// TIA Portal project "FactoryIO_Template_S7-1500_V15_V16_V17" (V17)

(* hardware
DEVICE "S71500/ET200MP-Station_1"  S7-1500 station
   slot 0: "Profilschiene_0"  6ES7 590-1***0-0AA0
   slot 1: "PLC_1"  CPU 1511-1 PN  6ES7 511-1AK00-0AB0  V1.8
   slot 2: "DI 16x24VDC BA_1"  DI 16x24VDC BA  6ES7 521-1BH10-0AA0  V1.0
   slot 3: "DQ 32x24VDC/0.5A BA_1"  DQ 32x24VDC/0.5A BA  6ES7 522-1BL10-0AA0  V1.1
*)

// ===== PLC "PLC_1"  CPU 1511-1 PN =====

VAR_GLOBAL   // PLC tag table "Standard-Variablentabelle"
   "Tag_1" AT %E0.0 : Bool;
   "Tag_3" AT %E0.1 : Bool;
   "ALWAYS_FALSE" AT %M100.1 : Bool;
END_VAR

VAR_GLOBAL   // PLC tag table "R00_S01_DI"
   "PALLET_AT_ENTRY" AT %I10.0 : Bool;
   "PALLET_AT_EXIT" AT %I10.1 : Bool;
   "PALLET_LOADED" AT %I10.2 : Bool;
   "BOX_AT_ENTRY" AT %I10.3 : Bool;
   "PUSHER_LIMIT" AT %I10.4 : Bool;
   "PLATE_LIMIT" AT %I10.5 : Bool;
   "CLAMPED" AT %I10.6 : Bool;
   "ELEVATOR_MOVING" AT %I10.7 : Bool;
   "START" AT %I11.0 : Bool;
   "RESET" AT %I11.1 : Bool;
   "STOP" AT %I11.2 : Bool;
   "EMERGENCY_STOP" AT %I11.3 : Bool;
   "AUTO" AT %I11.4 : Bool;
   "FACTORY_IO_RUNING" AT %I11.5 : Bool;
END_VAR

VAR_GLOBAL   // PLC tag table "R00_S02_D0"
   "PALLET_FEEDER" AT %A0.0 : Bool;
   "LOAD_PALLET" AT %Q0.1 : Bool;
   "EXIT_CONVEYOR" AT %Q0.2 : Bool;
   "MOVE_TO_LIMIT" AT %Q0.3 : Bool;
   "ELEVATOR_UP" AT %Q0.4 : Bool;
   "ELEVATOR_DOWN" AT %Q0.5 : Bool;
   "BOX_FEEDER" AT %Q0.6 : Bool;
   "TURN" AT %Q0.7 : Bool;
   "PUSH" AT %Q1.0 : Bool;
   "LOAD_BELT" AT %Q1.1 : Bool;
   "CLAMP" AT %Q1.2 : Bool;
   "OPEN_PLATE" AT %Q1.3 : Bool;
   "WARNING_LIGHT" AT %Q1.4 : Bool;
   "START_LIGHT" AT %Q1.5 : Bool;
   "RESET_LIGHT" AT %Q1.6 : Bool;
   "STOP_LIGHT" AT %Q1.7 : Bool;
END_VAR

DATA_BLOCK "CONTADOR_CAJAS"   // DB2
{ S7_Optimized_Access := 'TRUE' }
VERSION : 0.1
   VAR
      RESET_CONTADOR_CAJAS_EN_FILA : Bool;
      FILA_COMPLETA : Bool;
      P_FILA_COMPLETA : Bool;
      RESET_NUM_FILAS : Bool;
      NIVEL_COMPLETO : Bool;
      P_NIVEL_COMPLETO : Bool;
      CANTIDAD_MAXIMA_NIVELES : Int := 4;
      RESET_NUM_NIVELES : Bool;
      CANTIDAD_MAXIMA_CAJAS_POR_FILA : Int := 3;
      CANTIDAD_MAXIMA_FILAS_POR_NIVEL : Int;
   END_VAR
BEGIN
END_DATA_BLOCK

DATA_BLOCK "PALETIZADORA_AUTOMATICO_DB"   // DB5
{ S7_Optimized_Access := 'TRUE' }
VERSION : 0.1
// stored: InstanceOfName PALETIZADORA_AUTOMATICO
"PALETIZADORA_AUTOMATICO"
BEGIN
END_DATA_BLOCK

// folder: System blocks/Program resources

DATA_BLOCK "CONTADOR_CAJAS_EN_FILA"   // DB1
{ S7_Optimized_Access := 'TRUE' }
AUTHOR : Simatic
FAMILY : IEC
NAME : CNTR
VERSION : 1.0
// stored: InstanceOfName IEC_COUNTER
"IEC_COUNTER"
BEGIN
END_DATA_BLOCK

DATA_BLOCK "CONTADOR_FILAS"   // DB3
{ S7_Optimized_Access := 'TRUE' }
AUTHOR : Simatic
FAMILY : IEC
NAME : CNTR
VERSION : 1.0
// stored: InstanceOfName IEC_COUNTER
"IEC_COUNTER"
BEGIN
END_DATA_BLOCK

DATA_BLOCK "CONTADOR_NIVELES"   // DB4
{ S7_Optimized_Access := 'TRUE' }
AUTHOR : Simatic
FAMILY : IEC
NAME : CNTR
VERSION : 1.0
// stored: InstanceOfName IEC_COUNTER
"IEC_COUNTER"
BEGIN
END_DATA_BLOCK

// folder: (top level)

FUNCTION_BLOCK "PALETIZADORA_AUTOMATICO"   // FB1, GRAPH_PLUS
{ S7_Optimized_Access := 'TRUE' }
VERSION : 0.1
   VAR_INPUT
      OFF_SQ : Bool := false;   // Turn sequence off
      INIT_SQ : Bool := false;   // Set sequence to initial state
      ACK_EF : Bool := false;   // Acknowledge all errors and faults
      S_PREV : Bool := false;   // Output previous step in parameter S_NO
      S_NEXT : Bool := false;   // Indicate next step in parameter S_NO
      SW_AUTO : Bool := false;   // Automatic mode
      SW_TAP : Bool := false;   // Semiautomatic/switch with transition
      SW_TOP : Bool := false;   // Semiautomatic/ignore transition
      SW_MAN : Bool := false;   // Manual mode
      S_SEL : Int := 0;   // Select step to be output to S_NO
      S_ON : Bool := false;   // Activate step indicated in S_NO
      S_OFF : Bool := false;   // Deactivate step indicated S_NO
      T_PUSH : Bool := false;   // Enable transition to switch in semi automatic mode
   END_VAR
   VAR_OUTPUT
      S_NO : Int := 0;   // Step number
      S_MORE : Bool := false;   // More steps are available and can be shown in S_NO
      S_ACTIVE : Bool := false;   // Step indicated in S_NO is active
      ERR_FLT : Bool := false;   // Interlock or supervision group error
      AUTO_ON : Bool := false;   // Automatic mode is active
      TAP_ON : Bool := false;   // Semiautomatic mode/step with transition enabled
      TOP_ON : Bool := false;   // Semiautomatic mode/ignore transition enabled
      MAN_ON : Bool := false;   // Manual mode is active
   END_VAR
   VAR
      HMI_INFO : Array[0..8] of UInt;
      IF_PAR : G7_IfParPlus_V2;
      RT_DATA : G7_RTDataPlus_V2;   // Internal data area
      Trans1 : G7_TransitionPlus_V2;   // Transition structure
      Trans2 : G7_TransitionPlus_V2;   // Transition structure
      Trans3 : G7_TransitionPlus_V2;   // Transition structure
      Trans4 : G7_TransitionPlus_V2;   // Transition structure
      Trans5 : G7_TransitionPlus_V2;   // Transition structure
      Trans6 : G7_TransitionPlus_V2;   // Transition structure
      Trans7 : G7_TransitionPlus_V2;   // Transition structure
      Trans8 : G7_TransitionPlus_V2;   // Transition structure
      Trans9 : G7_TransitionPlus_V2;   // Transition structure
      Trans10 : G7_TransitionPlus_V2;   // Transition structure
      Trans11 : G7_TransitionPlus_V2;   // Transition structure
      Trans12 : G7_TransitionPlus_V2;   // Transition structure
      Trans14 : G7_TransitionPlus_V2;   // Transition structure
      Trans13 : G7_TransitionPlus_V2;   // Transition structure
      Trans15 : G7_TransitionPlus_V2;   // Transition structure
      Trans16 : G7_TransitionPlus_V2;   // Transition structure
      Trans17 : G7_TransitionPlus_V2;   // Transition structure
      Trans18 : G7_TransitionPlus_V2;   // Transition structure
      Trans19 : G7_TransitionPlus_V2;   // Transition structure
      Trans20 : G7_TransitionPlus_V2;   // Transition structure
      START : G7_StepPlus_V2;   // Step structure
      LOAD_PALLET : G7_StepPlus_V2;   // Step structure
      STOP_PALLET : G7_StepPlus_V2;   // Step structure
      EL_UP_TO_TOP : G7_StepPlus_V2;   // Step structure
      BOX_FEEDER : G7_StepPlus_V2;   // Step structure
      WAIT_1 : G7_StepPlus_V2;   // Step structure
      PUSH_N_PART : G7_StepPlus_V2;   // Step structure
      INTER : G7_StepPlus_V2;   // Step structure
      N_FILAS_IMPAR : G7_StepPlus_V2;   // Step structure
      CLAMP : G7_StepPlus_V2;   // Step structure
      TURN_ON : G7_StepPlus_V2;   // Step structure
      TURN_OFF : G7_StepPlus_V2;   // Step structure
      OPENPLATE : G7_StepPlus_V2;   // Step structure
      ELEVATOR_DOWN : G7_StepPlus_V2;   // Step structure
      ELEVATOR_DOWN_TO_BOTTON : G7_StepPlus_V2;   // Step structure
      EXIT_CONVEYOR : G7_StepPlus_V2;   // Step structure
      SINI : Array[0..1] of USInt;
      LSTT : Array[0..19] of USInt;
      ATAJ : Array[0..19] of USInt;
      ATAB : Array[0..19] of USInt;
      PSTT : Array[0..19] of USInt;
      NSTT : Array[0..19] of USInt;
      ASSJ : Array[0..15] of USInt;
      ASSB : Array[0..15] of USInt;
      PTTS : Array[0..15] of USInt;
      NTTS : Array[0..15] of USInt;
      SW_SQTS : Array[0..15] of USInt;
      SWITCH : Array[0..6] of USInt;
      TVX : Array[0..9] of USInt;
      TTX : Array[0..9] of USInt;
      TSX : Array[0..1] of USInt;
      S00X : Array[0..1] of USInt;
      SOFFX : Array[0..1] of USInt;
      SONX : Array[0..1] of USInt;
      SAX : Array[0..1] of USInt;
      SERRX : Array[0..16] of USInt;
      SMX : Array[0..16] of USInt;
      S0X : Array[0..16] of USInt;
      S1X : Array[0..16] of USInt;
      IL_ALARM_INST : Program_Alarm;
      SUP_ALARM_INST : Program_Alarm;
      STEP_TIME_ALARM_INST : Program_Alarm;
      IEC_TIMER_INST : IEC_TIMER;
      TRANSACTION_FLAG : Bool := false;
   END_VAR
   // SINI[0] := 2;
   // LSTT[0] := 255;
   // LSTT[1] := 255;
   // LSTT[2] := 255;
   // LSTT[3] := 255;
   // LSTT[4] := 255;
   // LSTT[5] := 255;
   // LSTT[6] := 255;
   // LSTT[8] := 255;
   // LSTT[9] := 4;
   // LSTT[10] := 255;
   // LSTT[11] := 255;
   // LSTT[12] := 255;
   // LSTT[13] := 255;
   // LSTT[14] := 255;
   // LSTT[15] := 255;
   // LSTT[16] := 4;
   // LSTT[17] := 255;
   // LSTT[18] := 255;
   // ATAJ[1] := 1;
   // ATAJ[2] := 2;
   // ATAJ[3] := 3;
   // ATAJ[4] := 4;
   // ATAJ[5] := 5;
   // ATAJ[6] := 6;
   // ATAJ[7] := 7;
   // ATAJ[8] := 8;
   // ATAJ[9] := 9;
   // ATAJ[10] := 10;
   // ATAJ[11] := 11;
   // ATAJ[12] := 12;
   // ATAJ[13] := 14;
   // ATAJ[14] := 13;
   // ATAJ[15] := 15;
   // ATAJ[16] := 16;
   // ATAJ[17] := 17;
   // ATAJ[18] := 18;
   // ATAJ[19] := 19;
   // ATAB[1] := 1;
   // ATAB[2] := 2;
   // ATAB[3] := 3;
   // ATAB[4] := 4;
   // ATAB[5] := 5;
   // ATAB[6] := 6;
   // ATAB[7] := 8;
   // ATAB[8] := 7;
   // ATAB[9] := 10;
   // ATAB[10] := 9;
   // ATAB[11] := 12;
   // ATAB[12] := 11;
   // ATAB[13] := 13;
   // ATAB[14] := 14;
   // ATAB[15] := 15;
   // ATAB[16] := 17;
   // ATAB[17] := 16;
   // ATAB[18] := 18;
   // ATAB[19] := 19;
   // PSTT[1] := 1;
   // PSTT[2] := 2;
   // PSTT[3] := 3;
   // PSTT[4] := 4;
   // PSTT[5] := 5;
   // PSTT[6] := 6;
   // PSTT[7] := 7;
   // PSTT[8] := 7;
   // PSTT[9] := 8;
   // PSTT[10] := 8;
   // PSTT[11] := 9;
   // PSTT[12] := 9;
   // PSTT[13] := 10;
   // PSTT[14] := 11;
   // PSTT[15] := 12;
   // PSTT[16] := 13;
   // PSTT[17] := 13;
   // PSTT[18] := 14;
   // PSTT[19] := 15;
   // NSTT[0] := 1;
   // NSTT[1] := 2;
   // NSTT[2] := 3;
   // NSTT[3] := 4;
   // NSTT[4] := 5;
   // NSTT[5] := 6;
   // NSTT[6] := 7;
   // NSTT[8] := 8;
   // NSTT[9] := 4;
   // NSTT[10] := 9;
   // NSTT[11] := 10;
   // NSTT[12] := 11;
   // NSTT[13] := 12;
   // NSTT[14] := 12;
   // NSTT[15] := 13;
   // NSTT[16] := 4;
   // NSTT[17] := 14;
   // NSTT[18] := 15;
   // ASSJ[1] := 1;
   // ASSJ[2] := 2;
   // ASSJ[3] := 3;
   // ASSJ[4] := 4;
   // ASSJ[5] := 5;
   // ASSJ[6] := 6;
   // ASSJ[7] := 7;
   // ASSJ[8] := 8;
   // ASSJ[9] := 9;
   // ASSJ[10] := 10;
   // ASSJ[11] := 11;
   // ASSJ[12] := 12;
   // ASSJ[13] := 13;
   // ASSJ[14] := 14;
   // ASSJ[15] := 15;
   // ASSB[1] := 1;
   // ASSB[2] := 2;
   // ASSB[3] := 3;
   // ASSB[4] := 4;
   // ASSB[5] := 5;
   // ASSB[6] := 6;
   // ASSB[7] := 7;
   // ASSB[8] := 8;
   // ASSB[9] := 9;
   // ASSB[10] := 10;
   // ASSB[11] := 11;
   // ASSB[12] := 12;
   // ASSB[13] := 13;
   // ASSB[14] := 14;
   // ASSB[15] := 15;
   // PTTS[0] := 255;
   // PTTS[2] := 1;
   // PTTS[3] := 2;
   // PTTS[4] := 3;
   // PTTS[5] := 4;
   // PTTS[6] := 5;
   // PTTS[7] := 6;
   // PTTS[8] := 8;
   // PTTS[9] := 10;
   // PTTS[10] := 11;
   // PTTS[11] := 12;
   // PTTS[12] := 13;
   // PTTS[13] := 15;
   // PTTS[14] := 17;
   // PTTS[15] := 18;
   // NTTS[1] := 1;
   // NTTS[2] := 2;
   // NTTS[3] := 3;
   // NTTS[4] := 4;
   // NTTS[5] := 5;
   // NTTS[6] := 6;
   // NTTS[7] := 7;
   // NTTS[8] := 9;
   // NTTS[9] := 11;
   // NTTS[10] := 13;
   // NTTS[11] := 14;
   // NTTS[12] := 15;
   // NTTS[13] := 16;
   // NTTS[14] := 18;
   // NTTS[15] := 19;
   // SW_SQTS[8] := 1;
   // SW_SQTS[9] := 2;
   // SW_SQTS[10] := 3;
   // SW_SQTS[11] := 4;
   // SW_SQTS[12] := 5;
   // SW_SQTS[13] := 5;
   // SW_SQTS[14] := 6;
   // SW_SQTS[15] := 6;
   // TVX[0] := 16#1;
   // TTX[0] := 16#1;
   // TSX[0] := 16#1;
   // S00X[0] := 16#1;
   // SOFFX[0] := 16#1;
   // SONX[0] := 16#1;
   // SAX[0] := 16#1;
   // SERRX[0] := 16#1;
   // SMX[0] := 16#1;
   // S0X[0] := 16#1;
   // S1X[0] := 16#1;
BEGIN
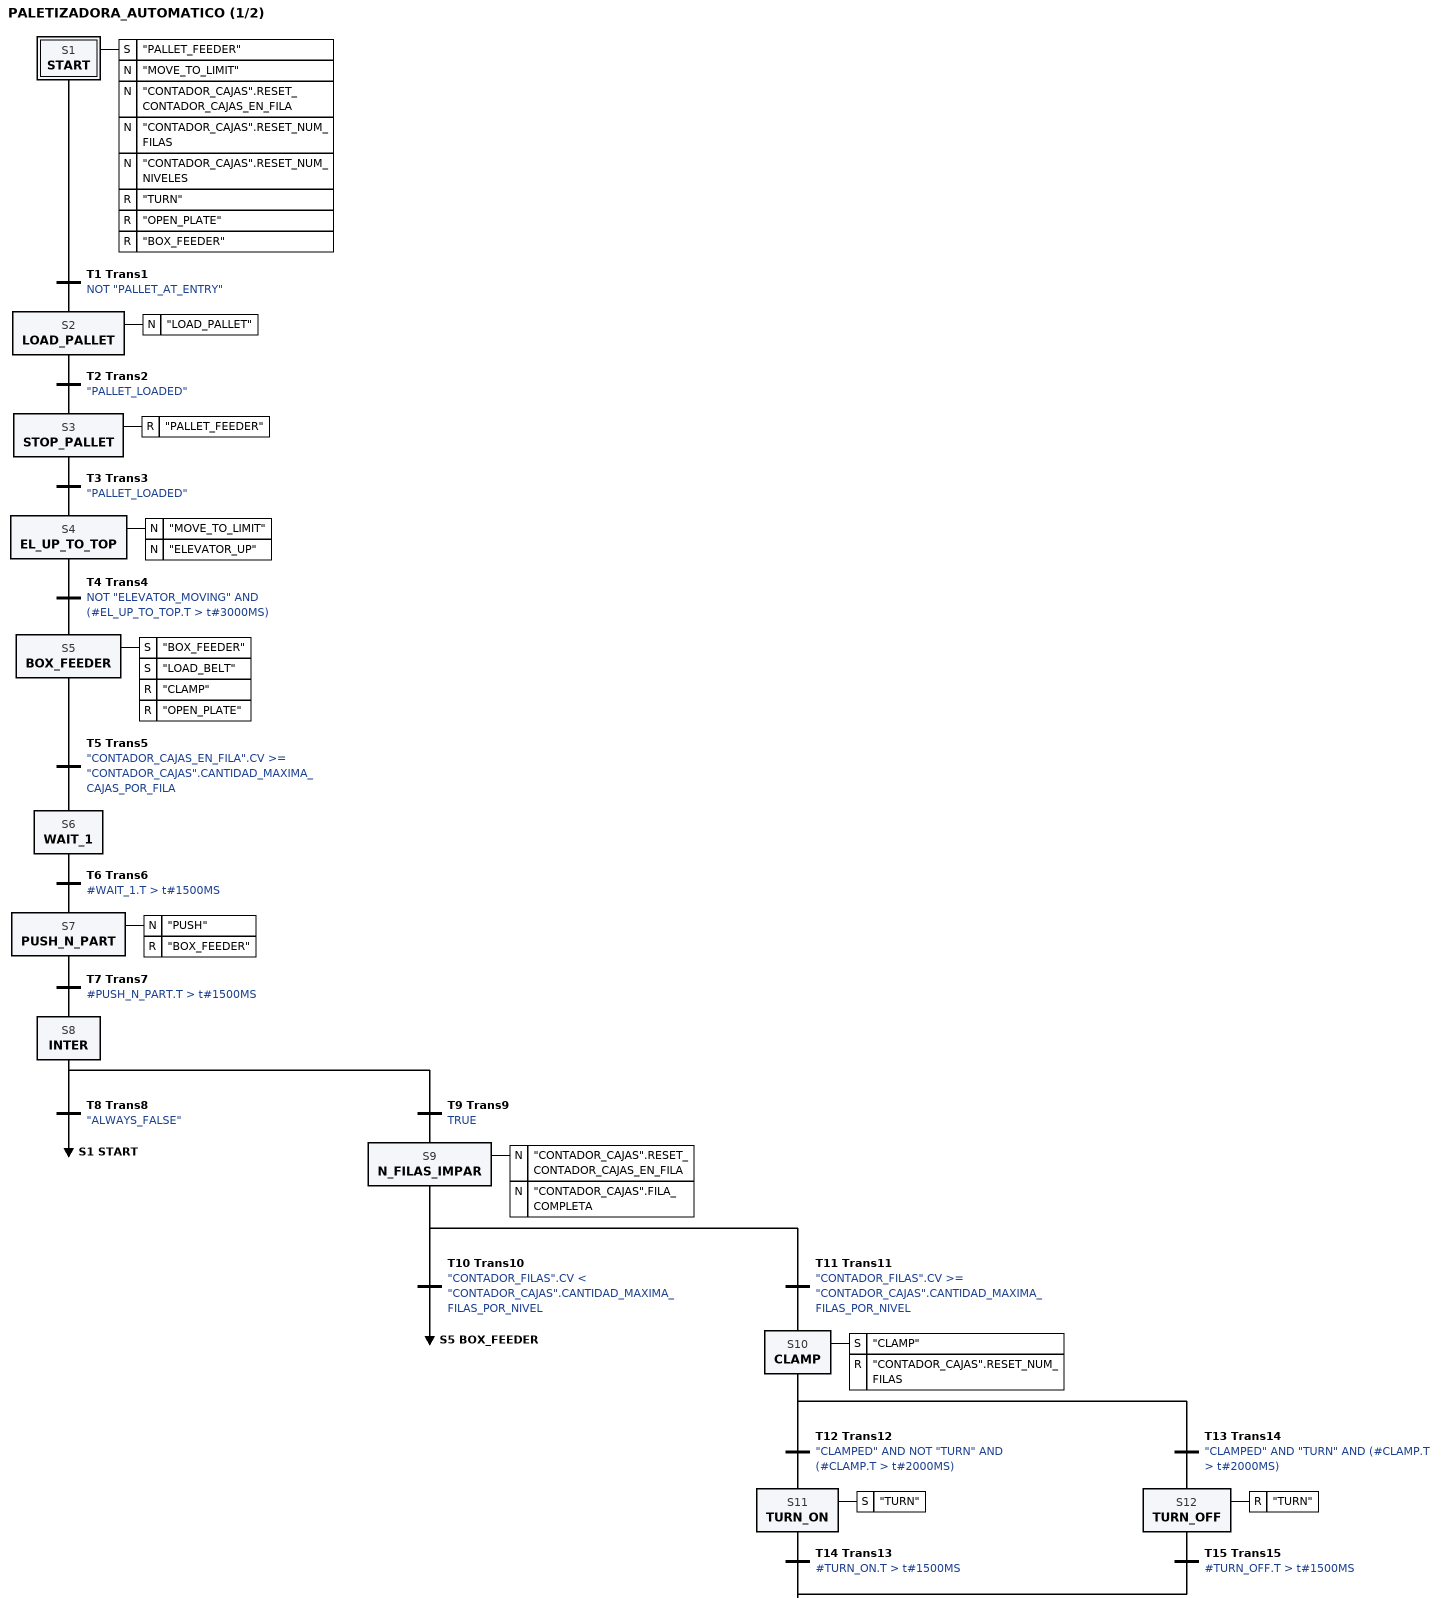
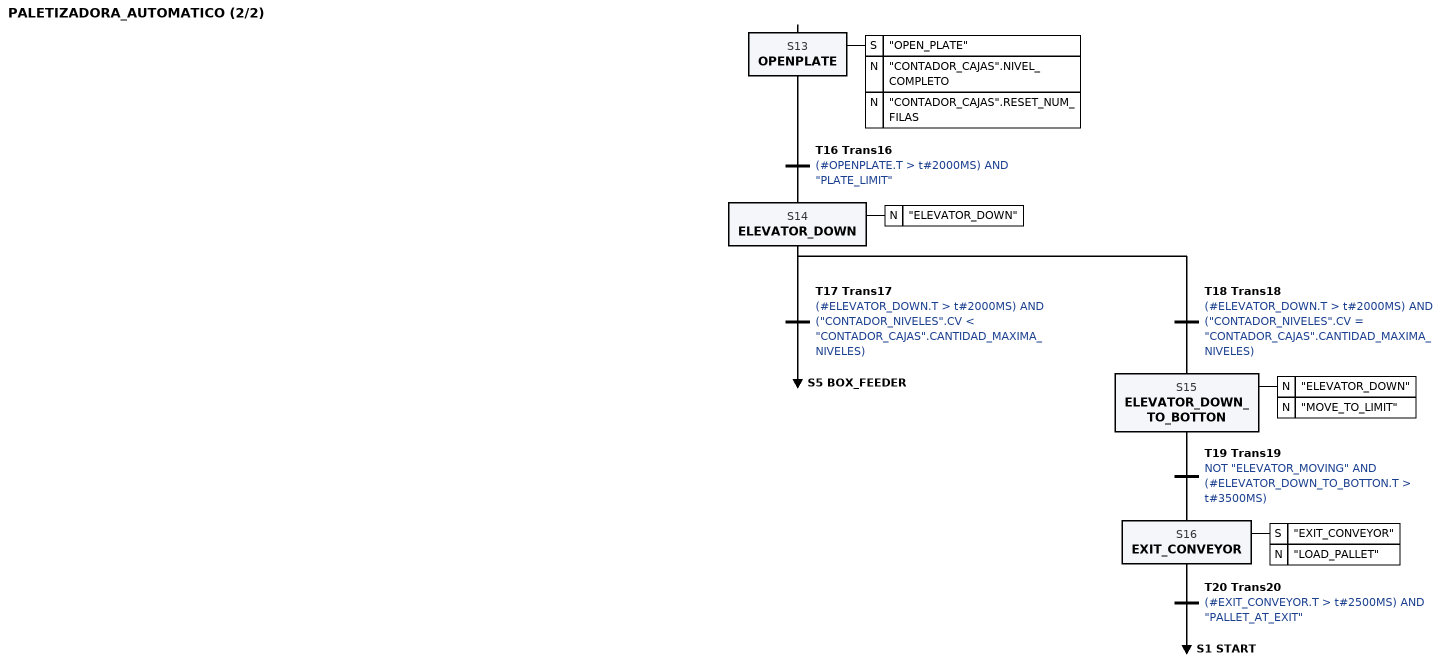
   // sequencer 1
   INITIAL_STEP START:   // S1, max time T#10S, warning time T#7S
              S    "PALLET_FEEDER"
              N    "MOVE_TO_LIMIT"
              N    "CONTADOR_CAJAS".RESET_CONTADOR_CAJAS_EN_FILA
              N    "CONTADOR_CAJAS".RESET_NUM_FILAS
              N    "CONTADOR_CAJAS".RESET_NUM_NIVELES
              R    "TURN"
              R    "OPEN_PLATE"
              R    "BOX_FEEDER"
   END_STEP
   TRANSITION Trans1 FROM START TO LOAD_PALLET   // T1
      := NOT "PALLET_AT_ENTRY";
   END_TRANSITION
   STEP LOAD_PALLET:   // S2, max time T#10S, warning time T#7S
              N    "LOAD_PALLET"
   END_STEP
   TRANSITION Trans2 FROM LOAD_PALLET TO STOP_PALLET   // T2
      := "PALLET_LOADED";
   END_TRANSITION
   STEP STOP_PALLET:   // S3, max time T#10S, warning time T#7S
              R    "PALLET_FEEDER"
   END_STEP
   TRANSITION Trans3 FROM STOP_PALLET TO EL_UP_TO_TOP   // T3
      := "PALLET_LOADED";
   END_TRANSITION
   STEP EL_UP_TO_TOP:   // S4, max time T#10S, warning time T#7S
              N    "MOVE_TO_LIMIT"
              N    "ELEVATOR_UP"
   END_STEP
   TRANSITION Trans4 FROM EL_UP_TO_TOP TO BOX_FEEDER   // T4
      := NOT "ELEVATOR_MOVING" AND (#EL_UP_TO_TOP.T > t#3000MS);
   END_TRANSITION
   STEP BOX_FEEDER:   // S5, max time T#10S, warning time T#7S
              S    "BOX_FEEDER"
              S    "LOAD_BELT"
              R    "CLAMP"
              R    "OPEN_PLATE"
   END_STEP
   TRANSITION Trans5 FROM BOX_FEEDER TO WAIT_1   // T5
      := "CONTADOR_CAJAS_EN_FILA".CV >= "CONTADOR_CAJAS".CANTIDAD_MAXIMA_CAJAS_POR_FILA;
   END_TRANSITION
   STEP WAIT_1:   // S6, max time T#10S, warning time T#7S
   END_STEP
   TRANSITION Trans6 FROM WAIT_1 TO PUSH_N_PART   // T6
      := #WAIT_1.T > t#1500MS;
   END_TRANSITION
   STEP PUSH_N_PART:   // S7, max time T#10S, warning time T#7S
              N    "PUSH"
              R    "BOX_FEEDER"
   END_STEP
   TRANSITION Trans7 FROM PUSH_N_PART TO INTER   // T7
      := #PUSH_N_PART.T > t#1500MS;
   END_TRANSITION
   STEP INTER:   // S8, max time T#10S, warning time T#7S
   END_STEP
   TRANSITION Trans8 FROM INTER TO START   // T8, jump
      := "ALWAYS_FALSE";
   END_TRANSITION
   TRANSITION Trans9 FROM INTER TO N_FILAS_IMPAR   // T9
      := TRUE;
   END_TRANSITION
   STEP N_FILAS_IMPAR:   // S9, max time T#10S, warning time T#7S
              N    "CONTADOR_CAJAS".RESET_CONTADOR_CAJAS_EN_FILA
              N    "CONTADOR_CAJAS".FILA_COMPLETA
   END_STEP
   TRANSITION Trans10 FROM N_FILAS_IMPAR TO BOX_FEEDER   // T10, jump
      := "CONTADOR_FILAS".CV < "CONTADOR_CAJAS".CANTIDAD_MAXIMA_FILAS_POR_NIVEL;
   END_TRANSITION
   TRANSITION Trans11 FROM N_FILAS_IMPAR TO CLAMP   // T11
      := "CONTADOR_FILAS".CV >= "CONTADOR_CAJAS".CANTIDAD_MAXIMA_FILAS_POR_NIVEL;
   END_TRANSITION
   STEP CLAMP:   // S10, max time T#10S, warning time T#7S
              S    "CLAMP"
              R    "CONTADOR_CAJAS".RESET_NUM_FILAS
   END_STEP
   TRANSITION Trans12 FROM CLAMP TO TURN_ON   // T12
      := "CLAMPED" AND NOT "TURN" AND (#CLAMP.T > t#2000MS);
   END_TRANSITION
   TRANSITION Trans14 FROM CLAMP TO TURN_OFF   // T13
      := "CLAMPED" AND "TURN" AND (#CLAMP.T > t#2000MS);
   END_TRANSITION
   STEP TURN_ON:   // S11, max time T#10S, warning time T#7S
              S    "TURN"
   END_STEP
   TRANSITION Trans13 FROM TURN_ON TO OPENPLATE   // T14
      := #TURN_ON.T > t#1500MS;
   END_TRANSITION
   STEP TURN_OFF:   // S12, max time T#10S, warning time T#7S
              R    "TURN"
   END_STEP
   TRANSITION Trans15 FROM TURN_OFF TO OPENPLATE   // T15
      := #TURN_OFF.T > t#1500MS;
   END_TRANSITION
   STEP OPENPLATE:   // S13, max time T#10S, warning time T#7S
              S    "OPEN_PLATE"
              N    "CONTADOR_CAJAS".NIVEL_COMPLETO
              N    "CONTADOR_CAJAS".RESET_NUM_FILAS
   END_STEP
   TRANSITION Trans16 FROM OPENPLATE TO ELEVATOR_DOWN   // T16
      := (#OPENPLATE.T > t#2000MS) AND "PLATE_LIMIT";
   END_TRANSITION
   STEP ELEVATOR_DOWN:   // S14, max time T#10S, warning time T#7S
              N    "ELEVATOR_DOWN"
   END_STEP
   TRANSITION Trans17 FROM ELEVATOR_DOWN TO BOX_FEEDER   // T17, jump
      := (#ELEVATOR_DOWN.T > t#2000MS) AND ("CONTADOR_NIVELES".CV < "CONTADOR_CAJAS".CANTIDAD_MAXIMA_NIVELES);
   END_TRANSITION
   TRANSITION Trans18 FROM ELEVATOR_DOWN TO ELEVATOR_DOWN_TO_BOTTON   // T18
      := (#ELEVATOR_DOWN.T > t#2000MS) AND ("CONTADOR_NIVELES".CV = "CONTADOR_CAJAS".CANTIDAD_MAXIMA_NIVELES);
   END_TRANSITION
   STEP ELEVATOR_DOWN_TO_BOTTON:   // S15, max time T#10S, warning time T#7S
              N    "ELEVATOR_DOWN"
              N    "MOVE_TO_LIMIT"
   END_STEP
   TRANSITION Trans19 FROM ELEVATOR_DOWN_TO_BOTTON TO EXIT_CONVEYOR   // T19
      := NOT "ELEVATOR_MOVING" AND (#ELEVATOR_DOWN_TO_BOTTON.T > t#3500MS);
   END_TRANSITION
   STEP EXIT_CONVEYOR:   // S16, max time T#10S, warning time T#7S
              S    "EXIT_CONVEYOR"
              N    "LOAD_PALLET"
   END_STEP
   TRANSITION Trans20 FROM EXIT_CONVEYOR TO START   // T20, jump
      := (#EXIT_CONVEYOR.T > t#2500MS) AND "PALLET_AT_EXIT";
   END_TRANSITION
END_FUNCTION_BLOCK

FUNCTION "BOX_COUNTER" : Void   // FC1, LAD
{ S7_Optimized_Access := 'TRUE' }
VERSION : 0.1
   VAR_TEMP   // added for the SCL form of the ladder/FBD networks
      _w1 : Bool;
   END_VAR
BEGIN

REGION Network 1: CONTADOR DE CAJAS
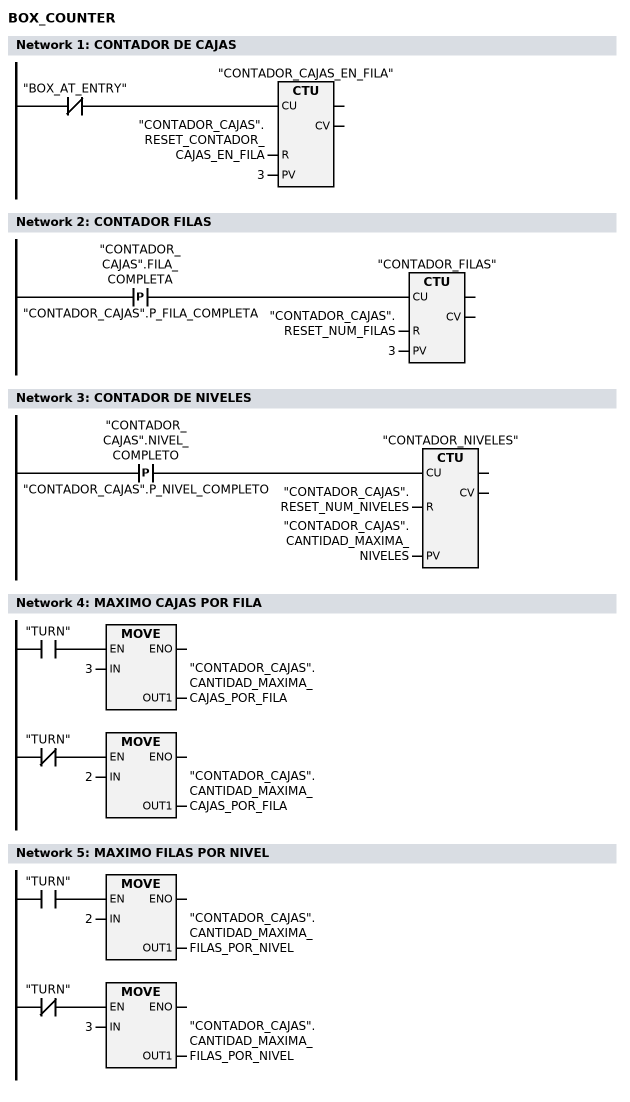
   "CONTADOR_CAJAS_EN_FILA".CTU(CU := NOT "BOX_AT_ENTRY",
                           R := "CONTADOR_CAJAS".RESET_CONTADOR_CAJAS_EN_FILA,
                           PV := 3);
END_REGION

REGION Network 2: CONTADOR FILAS
   #_w1 := "CONTADOR_CAJAS".FILA_COMPLETA AND NOT "CONTADOR_CAJAS".P_FILA_COMPLETA;   // rising edge of "CONTADOR_CAJAS".FILA_COMPLETA
   "CONTADOR_CAJAS".P_FILA_COMPLETA := "CONTADOR_CAJAS".FILA_COMPLETA;
   "CONTADOR_FILAS".CTU(CU := #_w1, R := "CONTADOR_CAJAS".RESET_NUM_FILAS, PV := 3);
END_REGION

REGION Network 3: CONTADOR DE NIVELES
   #_w1 := "CONTADOR_CAJAS".NIVEL_COMPLETO AND NOT "CONTADOR_CAJAS".P_NIVEL_COMPLETO;   // rising edge of "CONTADOR_CAJAS".NIVEL_COMPLETO
   "CONTADOR_CAJAS".P_NIVEL_COMPLETO := "CONTADOR_CAJAS".NIVEL_COMPLETO;
   "CONTADOR_NIVELES".CTU(CU := #_w1,
                          R := "CONTADOR_CAJAS".RESET_NUM_NIVELES,
                          PV := "CONTADOR_CAJAS".CANTIDAD_MAXIMA_NIVELES);
END_REGION

REGION Network 4: MAXIMO CAJAS POR FILA
   RUNG wire#powerrail
      Contact( "TURN" )
      Move(in := 3, out1 => "CONTADOR_CAJAS".CANTIDAD_MAXIMA_CAJAS_POR_FILA)
   END_RUNG
   RUNG wire#powerrail
      I_Contact( "TURN" )
      Move(in := 2, out1 => "CONTADOR_CAJAS".CANTIDAD_MAXIMA_CAJAS_POR_FILA)
   END_RUNG
   // the same network as SCL:
   IF "TURN" THEN "CONTADOR_CAJAS".CANTIDAD_MAXIMA_CAJAS_POR_FILA := 3; END_IF;
   IF NOT "TURN" THEN "CONTADOR_CAJAS".CANTIDAD_MAXIMA_CAJAS_POR_FILA := 2; END_IF;
END_REGION

REGION Network 5: MAXIMO FILAS POR NIVEL
   RUNG wire#powerrail
      Contact( "TURN" )
      Move(in := 2, out1 => "CONTADOR_CAJAS".CANTIDAD_MAXIMA_FILAS_POR_NIVEL)
   END_RUNG
   RUNG wire#powerrail
      I_Contact( "TURN" )
      Move(in := 3, out1 => "CONTADOR_CAJAS".CANTIDAD_MAXIMA_FILAS_POR_NIVEL)
   END_RUNG
   // the same network as SCL:
   IF "TURN" THEN "CONTADOR_CAJAS".CANTIDAD_MAXIMA_FILAS_POR_NIVEL := 2; END_IF;
   IF NOT "TURN" THEN "CONTADOR_CAJAS".CANTIDAD_MAXIMA_FILAS_POR_NIVEL := 3; END_IF;
END_REGION
END_FUNCTION

FUNCTION "MHJ-PLC-Lab-Function-S71500" : Void   // FC9000, SCL
{ S7_Optimized_Access := 'TRUE' }
VERSION : 0.1
   VAR_TEMP
      Value : Byte;
      ForCounter : Int;
   END_VAR
   VAR CONSTANT
      Value_01_DW : DWord := 16#1223_5486;
      Value_02_DW : DWord := 16#A6C9_D1F5;
   END_VAR
BEGIN

   #Value:=PEEK(area := 16#82,
        dbNumber := 0,
        byteOffset := 511);
   #Value := #Value + 1;

   POKE(area := 16#82,
        dbNumber := 0,
        byteOffset := 511,
        value := #Value);

   POKE(area := 16#82,
        dbNumber := 0,
        byteOffset := 1016,
        value := #Value_01_DW);
   POKE(area := 16#82,
        dbNumber := 0,
        byteOffset := 1020,
        value := #Value_02_DW);

   FOR #ForCounter := 0 TO 63 DO
       #Value:=PEEK(area := 16#1,
            dbNumber := 0,
            byteOffset := #ForCounter);
       POKE(area := 16#81,
            dbNumber := 0,
            byteOffset := #ForCounter,
            value := #Value);
   END_FOR;
   #Value := PEEK(area := 16#1,
                  dbNumber := 0,
                  byteOffset := 512);
   POKE(area := 16#82,
        dbNumber := 0,
        byteOffset := 512,
        value := #Value);
END_FUNCTION

ORGANIZATION_BLOCK "Main"   // OB1, LAD, ProgramCycle
TITLE = "Main Program Sweep (Cycle)"
{ S7_Optimized_Access := 'TRUE' }
VERSION : 0.1
   VAR_INPUT
      Initial_Call : Bool;   // Initial call of this OB
      Remanence : Bool;   // =True, if remanent data are available
   END_VAR
BEGIN

REGION Network 1
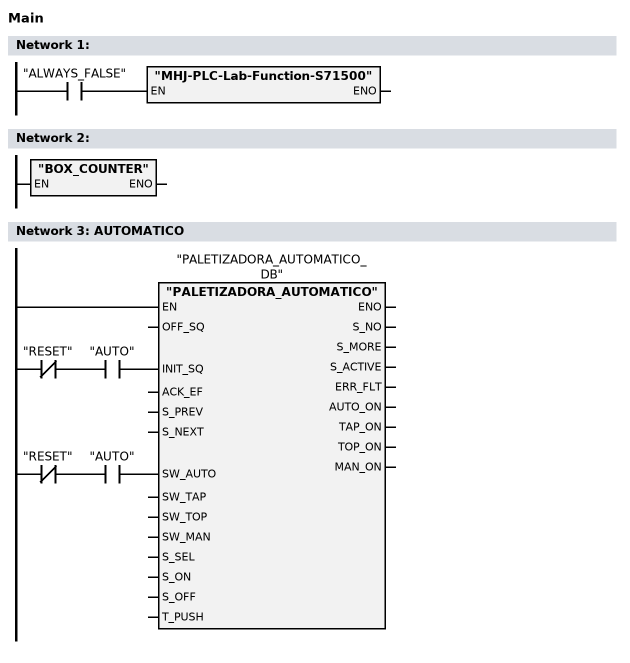
   RUNG wire#powerrail
      Contact( "ALWAYS_FALSE" )
      "MHJ-PLC-Lab-Function-S71500"()
   END_RUNG
   // the same network as SCL:
   IF "ALWAYS_FALSE" THEN "MHJ-PLC-Lab-Function-S71500"(); END_IF;
END_REGION

REGION Network 2
   RUNG wire#powerrail
      "BOX_COUNTER"()
   END_RUNG
   // the same network as SCL:
   "BOX_COUNTER"();
END_REGION

REGION Network 3: AUTOMATICO
   RUNG wire#powerrail
      "PALETIZADORA_AUTOMATICO_DB"(INIT_SQ := wire#w1, SW_AUTO := wire#w2, OFF_SQ :=, ACK_EF :=, S_PREV :=, S_NEXT :=, SW_TAP :=, SW_TOP :=, SW_MAN :=, S_SEL :=, S_ON :=, S_OFF :=, T_PUSH :=, S_NO =>, S_MORE =>, S_ACTIVE =>, ERR_FLT =>, AUTO_ON =>, TAP_ON =>, TOP_ON =>, MAN_ON =>)
   END_RUNG
   RUNG wire#powerrail
      I_Contact( "RESET" )
      Contact( "AUTO" )
   END_RUNG wire#w1
   RUNG wire#powerrail
      I_Contact( "RESET" )
      Contact( "AUTO" )
   END_RUNG wire#w2
   // the same network as SCL:
   "PALETIZADORA_AUTOMATICO_DB"(INIT_SQ := NOT "RESET" AND "AUTO", SW_AUTO := NOT "RESET" AND "AUTO");   // "PALETIZADORA_AUTOMATICO"
END_REGION
END_ORGANIZATION_BLOCK